Yaskawa INFORM job: pipe_reducer_cylinder_program.JBI

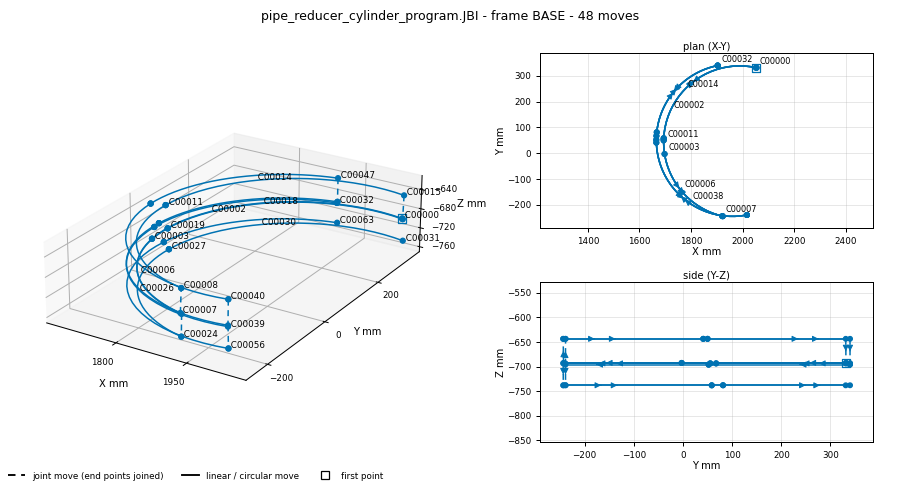
[picture p0: tool path of pipe_reducer_cylinder_program.JBI in frame BASE, 48 of 69 moves have a stored position in this frame; points joined in program order, loops and branches not executed]
/JOB
//NAME pipe_reducer_cylinder_program
//POS
///NPOS 64,0,64,0,0,0
///TOOL 0
///POSTYPE BASE
///RECTAN
///RCONF 0,0,0,0,0,0,0,0,0,0,0,0,0,0,0,0,0,0,0,0,0,0,0,0
C00000=2050.805847,331.670968,-692.358000,77.782541,-90.000000,5.000000
C00001=2050.805847,331.670968,-692.358000,77.782541,-90.000000,5.000000
C00002=1718.426807,161.905790,-692.358000,156.329511,-89.999999,5.000000
C00003=1697.289395,-2.780256,-692.358000,-170.957335,-89.999999,5.000000
C00004=1697.289395,-2.780256,-692.358000,-170.957335,-89.999999,5.000000
C00005=1697.289395,-2.780256,-692.358000,-170.957335,-89.999999,5.000000
C00006=1761.870554,-145.071816,-692.358000,-140.219395,-90.000000,5.000000
C00007=1919.652971,-243.109369,-692.358000,-103.489818,-90.000000,5.000000
C00008=1922.450580,-243.766086,-643.405460,175.000000,-60.000000,77.068702
C00009=1922.450580,-243.766086,-643.405460,175.000000,-60.000000,77.068702
C00010=1750.661125,-130.730297,-643.405460,175.000000,-60.000000,36.242244
C00011=1693.694756,49.939644,-643.405460,175.000000,-60.000000,-5.000000
C00012=1693.694756,49.939644,-643.405460,175.000000,-60.000000,-5.000000
C00013=1693.694756,49.939644,-643.405460,175.000000,-60.000000,-5.000000
C00014=1772.082682,243.807522,-643.405460,175.000000,-60.000000,-42.789134
C00015=2053.518341,331.070247,-643.405460,175.000000,-60.000000,-102.757430
C00016=2051.873274,331.437771,-693.362960,-175.000000,-60.000000,-102.429815
C00017=2051.873274,331.437771,-693.362960,-175.000000,-60.000000,-102.429815
C00018=1780.545668,252.579253,-693.362960,-175.000000,-60.000000,-45.158283
C00019=1693.864969,55.431086,-693.362960,175.000000,-60.000000,-5.000000
C00020=1693.864969,55.431086,-693.362960,175.000000,-60.000000,-5.000000
C00021=1693.864969,55.431086,-693.362960,175.000000,-60.000000,-5.000000
C00022=1751.570168,-131.963691,-693.362960,175.000000,-60.000000,36.540038
C00023=1922.676560,-243.817879,-693.362960,-175.000000,-60.000000,77.113762
C00024=1921.350884,-243.511373,-737.979960,-175.000000,-60.000000,76.849309
C00025=1921.350884,-243.511373,-737.979960,-175.000000,-60.000000,76.849309
C00026=1748.830985,-128.205697,-737.979960,175.000000,-60.000000,35.636198
C00027=1694.002932,58.464173,-737.979960,-175.000000,-60.000000,-5.000000
C00028=1694.002932,58.464173,-737.979960,-175.000000,-60.000000,-5.000000
C00029=1694.002932,58.464173,-737.979960,-175.000000,-60.000000,-5.000000
C00030=1777.876037,249.889983,-737.979960,175.000000,-60.000000,-44.421789
C00031=2053.964411,330.968887,-737.979960,175.000000,-60.000000,-102.846337
C00032=1902.219665,339.515195,-695.854500,101.326687,-90.000000,5.000000
C00033=1902.219665,339.515195,-695.854500,101.326687,-90.000000,5.000000
C00034=1732.354711,237.619152,-695.854500,140.589451,-90.000000,5.000000
C00035=1665.328035,52.141306,-695.854500,175.000000,-89.999999,5.000000
C00036=1665.328035,52.141306,-695.854500,175.000000,-89.999999,5.000000
C00037=1665.328035,52.141306,-695.854500,175.000000,-89.999999,5.000000
C00038=1790.172366,-190.416743,-695.854500,-125.203929,-89.999999,5.000000
C00039=2015.458581,-239.092203,-695.854500,-79.179965,-90.000000,5.000000
C00040=2016.240040,-238.941755,-643.407460,175.000000,-60.000000,100.974707
C00041=2016.240040,-238.941755,-643.407460,175.000000,-60.000000,100.974707
C00042=1774.182996,-178.300430,-643.407460,175.000000,-60.000000,50.896198
C00043=1665.470521,41.144783,-643.407460,175.000000,-60.000000,5.000000
C00044=1665.470521,41.144783,-643.407460,175.000000,-60.000000,5.000000
C00045=1665.470521,41.144783,-643.407460,175.000000,-60.000000,5.000000
C00046=1747.257077,254.408426,-643.407460,-175.000000,-60.000000,-43.774759
C00047=1903.464598,339.761774,-643.407460,-175.000000,-60.000000,-78.919976
C00048=1903.271014,339.723797,-693.377460,175.000000,-60.000000,-78.881634
C00049=1903.271014,339.723797,-693.377460,175.000000,-60.000000,-78.881634
C00050=1754.819723,262.019406,-693.377460,175.000000,-60.000000,-45.860225
C00051=1665.804513,67.299765,-693.377460,175.000000,-60.000000,-5.000000
C00052=1665.804513,67.299765,-693.377460,175.000000,-60.000000,-5.000000
C00053=1665.804513,67.299765,-693.377460,175.000000,-60.000000,-5.000000
C00054=1765.688937,-171.126375,-693.377460,175.000000,-60.000000,48.735143
C00055=2015.601917,-239.064771,-693.377460,175.000000,-60.000000,100.848400
C00056=2016.274218,-238.935125,-737.875460,-175.000000,-60.000000,100.981474
C00057=2016.274218,-238.935125,-737.875460,-175.000000,-60.000000,100.981474
C00058=1755.316676,-161.576858,-737.875460,-175.000000,-60.000000,45.994661
C00059=1666.951480,81.402685,-737.875460,175.000000,-60.000000,-6.024700
C00060=1666.951480,81.402685,-737.875460,175.000000,-60.000000,-6.024700
C00061=1666.951480,81.402685,-737.875460,175.000000,-60.000000,-6.024700
C00062=1765.362383,271.763085,-737.875460,175.000000,-60.000000,-48.650652
C00063=1903.406265,339.750344,-737.875460,-175.000000,-60.000000,-78.908423
///POSTYPE PULSE
///PULSE
EX00000=78848.0
EX00001=287744.0
///POSTYPE PULSE
///PULSE
EC00000=78848.0
EC00001=78848.0
EC00002=78848.0
EC00003=78848.0
EC00004=78848.0
EC00005=78848.0
EC00006=78848.0
EC00007=78848.0
EC00008=78848.0
EC00009=78848.0
EC00010=78848.0
EC00011=78848.0
EC00012=78848.0
EC00013=78848.0
EC00014=78848.0
EC00015=78848.0
EC00016=78848.0
EC00017=78848.0
EC00018=78848.0
EC00019=78848.0
EC00020=78848.0
EC00021=78848.0
EC00022=78848.0
EC00023=78848.0
EC00024=78848.0
EC00025=78848.0
EC00026=78848.0
EC00027=78848.0
EC00028=78848.0
EC00029=78848.0
EC00030=78848.0
EC00031=78848.0
EC00032=287744.0
EC00033=287744.0
EC00034=287744.0
EC00035=287744.0
EC00036=287744.0
EC00037=287744.0
EC00038=287744.0
EC00039=287744.0
EC00040=287744.0
EC00041=287744.0
EC00042=287744.0
EC00043=287744.0
EC00044=287744.0
EC00045=287744.0
EC00046=287744.0
EC00047=287744.0
EC00048=287744.0
EC00049=287744.0
EC00050=287744.0
EC00051=287744.0
EC00052=287744.0
EC00053=287744.0
EC00054=287744.0
EC00055=287744.0
EC00056=287744.0
EC00057=287744.0
EC00058=287744.0
EC00059=287744.0
EC00060=287744.0
EC00061=287744.0
EC00062=287744.0
EC00063=287744.0
//INST
///DATE 2023/08/16 14:46
///ATTR SC,RW,RJ
////FRAME BASE
///GROUP1 RB1,ST1
NOP
MOVJ P009 EX000 VJ=15.00
MOVJ C00000 EC00000 VJ=15.0
CALL JOB:SPYON
MOVC C00001 EC00001 V=150.0
MOVC C00002 EC00002 V=150.0
MOVC C00003 EC00003 V=150.0
MOVJ C00004 EC00004 VJ=15.0
MOVC C00005 EC00005 V=150.0
MOVC C00006 EC00006 V=150.0
MOVC C00007 EC00007 V=150.0
MOVJ C00008 EC00008 VJ=15.0
MOVC C00009 EC00009 V=150.0
MOVC C00010 EC00010 V=150.0
MOVC C00011 EC00011 V=150.0
MOVJ C00012 EC00012 VJ=15.0
MOVC C00013 EC00013 V=150.0
MOVC C00014 EC00014 V=150.0
MOVC C00015 EC00015 V=150.0
MOVJ C00016 EC00016 VJ=15.0
MOVC C00017 EC00017 V=150.0
MOVC C00018 EC00018 V=150.0
MOVC C00019 EC00019 V=150.0
MOVJ C00020 EC00020 VJ=15.0
MOVC C00021 EC00021 V=150.0
MOVC C00022 EC00022 V=150.0
MOVC C00023 EC00023 V=150.0
MOVJ C00024 EC00024 VJ=15.0
MOVC C00025 EC00025 V=150.0
MOVC C00026 EC00026 V=150.0
MOVC C00027 EC00027 V=150.0
MOVJ C00028 EC00028 VJ=15.0
MOVC C00029 EC00029 V=150.0
MOVC C00030 EC00030 V=150.0
MOVC C00031 EC00031 V=150.0
CALL JOB:SPYOF
MOVJ P009 VJ=15.00
MOVL P009 EX00000 V=150.0
MOVJ C00032 EC00032 VJ=15.0
CALL JOB:SPYON
MOVC C00033 EC00033 V=150.0
MOVC C00034 EC00034 V=150.0
MOVC C00035 EC00035 V=150.0
MOVJ C00036 EC00036 VJ=15.0
MOVC C00037 EC00037 V=150.0
MOVC C00038 EC00038 V=150.0
MOVC C00039 EC00039 V=150.0
MOVJ C00040 EC00040 VJ=15.0
MOVC C00041 EC00041 V=150.0
MOVC C00042 EC00042 V=150.0
MOVC C00043 EC00043 V=150.0
MOVJ C00044 EC00044 VJ=15.0
MOVC C00045 EC00045 V=150.0
MOVC C00046 EC00046 V=150.0
MOVC C00047 EC00047 V=150.0
MOVJ C00048 EC00048 VJ=15.0
MOVC C00049 EC00049 V=150.0
MOVC C00050 EC00050 V=150.0
MOVC C00051 EC00051 V=150.0
MOVJ C00052 EC00052 VJ=15.0
MOVC C00053 EC00053 V=150.0
MOVC C00054 EC00054 V=150.0
MOVC C00055 EC00055 V=150.0
MOVJ C00056 EC00056 VJ=15.0
MOVC C00057 EC00057 V=150.0
MOVC C00058 EC00058 V=150.0
MOVC C00059 EC00059 V=150.0
MOVJ C00060 EC00060 VJ=15.0
MOVC C00061 EC00061 V=150.0
MOVC C00062 EC00062 V=150.0
MOVC C00063 EC00063 V=150.0
CALL JOB:SPYOF
MOVJ P009 VJ=15.00
MOVL P009 EX00001 V=150.0
END
